FUNCTION F_DRIVE_RESET : BOOL
VAR_INPUT
	timer_trigger: BOOL := FALSE;
END_VAR

VAR
END_VAR

IF timer_trigger THEN
	GVL.controlword_PLC_SLAVE := 16#80;
	GVL.tuning_cmd := 16#06;
ELSE
	GVL.controlword_PLC_SLAVE := GVL.controlword_PLC_NC;
END_IF
F_DRIVE_RESET := TRUE;

END_FUNCTION

(* stored: Version 1.1.0.1, ProductVersion 3.1.4022.16
   POU F_DRIVE_RESET: Id {2baa73a1-fc1d-45ef-85ef-d918f3c398b8}, SpecialFunc None *)
